Staubli VAL3: Control_BatPara.pgx

public program Control_BatPara(num x_nMax, num& x_nFrom[], num& x_nTo[], num& x_nValue[], bool& x_bEdit[])
  local string l_sItem[4]
  local num l_nNum
  local num l_nKey
  local num l_nData[6]
  local num l_nSelectIndex
  local string l_sS[5]
  local num l_nIndex
begin

  //为LasMAN3.7进行配置
  //批处理切割或者焊接点的参数
  //包括速度，加速度，blend, 工艺，动作




  x_bEdit[0]=x_bEdit[1]=x_bEdit[2]=x_bEdit[3]=x_bEdit[4]=false
  l_nData[0]=1
  l_nData[1]=x_nMax
  l_nData[2]=0
  l_nData[3]=1
  l_sS[0]="速度"
  l_sS[1]="加速度"
  l_sS[2]="Blend"
  l_sS[3]="工艺"
  l_sS[4]="动作"

  l_sItem[0]="开始序号:"+toString("",l_nData[0])
  l_sItem[1]="结束序号:"+toString("",l_nData[1])
  l_sItem[2]="选项    :"+l_sS[l_nData[2]]
  l_sItem[3]="值      :"+toString("",l_nData[3])



  call Control_BottomS(",,,,,,退出,修改")
  call Control_PanelXY(8,0,15,4)
  call Control_Panel("批处理参数")
  call Control_List(l_sItem,l_nSelectIndex)
  while true
    l_nKey=getKey()

    switch l_nKey
      case 261
        l_nSelectIndex=max(0,l_nSelectIndex-1)
      break

      case 266
        l_nSelectIndex=min(l_nSelectIndex+1,3)
      break

      case 278
        l_nIndex=round(min(max(0,l_nData[2]),4))
        x_nFrom[l_nIndex]=l_nData[0]
        x_nTo[l_nIndex]=l_nData[1]

        x_nValue[l_nIndex]=l_nData[3]
        x_bEdit[l_nIndex]=true
        popUpMsg(l_sS[l_nIndex]+"已修改")
       // cls()
        //return
      break


      case 277,255

        cls()
        //x_bEdit=false
        return
      break

      case 270
        if l_nSelectIndex==2
          call Sel_Edit(l_nData[2],nPanelLTopX+10,l_nSelectIndex+nPanelLTopY+1,l_sS)
        else
          call Float_Edit(l_nData[l_nSelectIndex],nPanelLTopX+10,l_nSelectIndex+nPanelLTopY+1)
          if l_nSelectIndex==0
            l_nData[l_nSelectIndex]=roundDown(min(l_nData[1],max(1,l_nData[l_nSelectIndex])))

          endIf
          if l_nSelectIndex==1
            l_nData[l_nSelectIndex]=roundDown(min(x_nMax,max(1,l_nData[l_nSelectIndex])))

          endIf
        endIf
      break


    endSwitch

    if l_nKey!=-1
      l_sItem[0]="开始序号:"+toString("",l_nData[0])
      l_sItem[1]="结束序号:"+toString("",l_nData[1])
      l_sItem[2]="选项    :"+l_sS[l_nData[2]]
      l_sItem[3]="值      :"+toString("",l_nData[3])

      call Control_List(l_sItem,l_nSelectIndex)

    endIf

  endWhile

end
